SUBAPPLICATION Uebung_022b_AX2 (* Spiegelabfolge (2) - AX Variante *)
  (* Standard: 61499-2; Description: Copyright (c) 2023 Meisterschulen am Ostbahnhof This program and the accompanying materials are made available under the terms of the Eclipse Public License 2.0 which is available at https://www.eclipse.org/legal/epl-2.0/ SPDX-License-Identifier: EPL-2.0 *)
  (* Version 1.0, 2026-04-20, Franz Höpfinger, Meisterschulen am Ostbahnhof, AX Variante *)
  PACKAGE Uebungen;
  IMPORT isobus::UT::io::Softkey::SoftKeyActivationCode::SK_PRESSED;
  IMPORT isobus::UT::io::Softkey::SoftKeyActivationCode::SK_RELEASED;
  IMPORT Uebungen::const::UT::DefaultPool::SoftKey_F1;
  IMPORT Uebungen::const::UT::DefaultPool::SoftKey_F2;
  IMPORT Uebungen::const::UT::DefaultPool::SoftKey_F3;
  IMPORT logiBUS::io::DQ::logiBUS_DO::Output_Q1;
  IMPORT logiBUS::io::DQ::logiBUS_DO::Output_Q2;
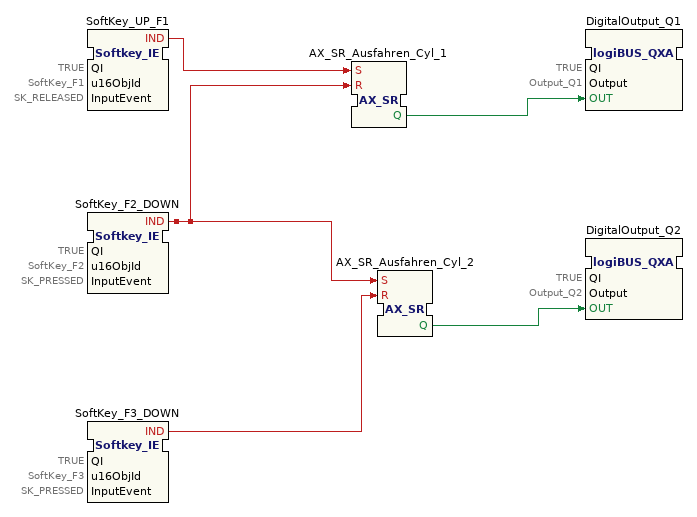
  (* START-Knopf *)
  (* Endlage Ausfahren_Cyl_1 *)
  (* Endlage Ausfahren_Cyl_2 *)
  (* Ausfahren_Cyl_1 *)
  (* Ausfahren_Cyl_2 *)
  FBS
    DigitalOutput_Q1 : logiBUS::io::DQ::logiBUS_QXA(QI := TRUE, Output := Output_Q1);
    SoftKey_UP_F1 : isobus::UT::io::Softkey::Softkey_IE(QI := TRUE, u16ObjId := SoftKey_F1, InputEvent := SK_RELEASED);
    AX_SR_Ausfahren_Cyl_1 : adapter::events::unidirectional::AX_SR;
    SoftKey_F2_DOWN : isobus::UT::io::Softkey::Softkey_IE(QI := TRUE, u16ObjId := SoftKey_F2, InputEvent := SK_PRESSED);
    DigitalOutput_Q2 : logiBUS::io::DQ::logiBUS_QXA(QI := TRUE, Output := Output_Q2);
    AX_SR_Ausfahren_Cyl_2 : adapter::events::unidirectional::AX_SR;
    SoftKey_F3_DOWN : isobus::UT::io::Softkey::Softkey_IE(QI := TRUE, u16ObjId := SoftKey_F3, InputEvent := SK_PRESSED);
  END_FBS
  EVENT_CONNECTIONS
    SoftKey_UP_F1.IND TO AX_SR_Ausfahren_Cyl_1.S;
    SoftKey_F2_DOWN.IND TO AX_SR_Ausfahren_Cyl_1.R;
    SoftKey_F2_DOWN.IND TO AX_SR_Ausfahren_Cyl_2.S;
    SoftKey_F3_DOWN.IND TO AX_SR_Ausfahren_Cyl_2.R;
  END_CONNECTIONS
  ADAPTER_CONNECTIONS
    AX_SR_Ausfahren_Cyl_1.Q TO DigitalOutput_Q1.OUT;
    AX_SR_Ausfahren_Cyl_2.Q TO DigitalOutput_Q2.OUT;
  END_CONNECTIONS
END_SUBAPPLICATION
